FUNCTION_BLOCK AI_Channel
VAR
	{attribute addProperty Name  "Raw value"}
	Value AT %I* : INT;
	Status AT %I* : AI_ChannelStatus;
END_VAR

END_FUNCTION_BLOCK

(* stored: Version 1.1.0.1, ProductVersion 3.1.4024.6
   POU AI_Channel: Id {ca9a68ab-d2b5-4a58-bd74-36e80f924e08}, SpecialFunc None *)
